(* IEC 61131-3 sources: GradProject/LadderLogic, 14 files *)

(* ---- Test10.st ---- *)
PROGRAM Test_Program
  VAR
    ESP0 AT %QX0.0 : BOOL;
  END_VAR
  VAR
    TMP : BOOL;
  END_VAR
  VAR
    ESP1 AT %QX0.1 : BOOL;
  END_VAR
  VAR
    TMP2 : BOOL;
    TMP4 : BOOL;
    TMP3 : BOOL;
    T0 : TOF;
    TON1 : TON;
    TON2 : TON;
    TON3 : TON;
  END_VAR

  T0(IN := NOT(TMP), PT := T#10000ms);
  ESP0 := T0.Q;
  TON1(IN := ESP0, PT := T#10000ms);
  ESP1 := TON1.Q;
  TON2(IN := ESP1, PT := T#10000ms);
  IF TON2.Q THEN
    ESP1 := FALSE; (*reset*)
  END_IF;
  TMP4 := NOT(TMP3);
  TON3(IN := TMP4, PT := T#30000ms);
  IF TON3.Q THEN
    ESP0 := FALSE; (*reset*)
  END_IF;
END_PROGRAM

CONFIGURATION Config0

  RESOURCE Res0 ON PLC
    TASK MyTask(INTERVAL := T#50ms,PRIORITY := 0);
    PROGRAM instance0 WITH MyTask : Test_Program;
  END_RESOURCE
END_CONFIGURATION

(* ---- Test11\.st ---- *)
PROGRAM Test_Program
  VAR
    ESP0 AT %QX0.0 : BOOL;
    TMP AT %QX1.3 : BOOL;
    ESP1 AT %QX0.1 : BOOL;
  END_VAR
  VAR
    TMP2 : BOOL;
    TMP4 : BOOL;
    TMP3 : BOOL;
    T0 : TOF;
    TON1 : TON;
    TON2 : TON;
    TON3 : TON;
  END_VAR

  T0(IN := TMP, PT := T#10000ms);
  ESP0 := T0.Q;
  TON1(IN := ESP0, PT := T#10000ms);
  ESP1 := TON1.Q;
  TON2(IN := ESP1, PT := T#10000ms);
  IF TON2.Q THEN
    ESP1 := FALSE; (*reset*)
  END_IF;
  TMP4 := NOT(TMP3);
  TON3(IN := TMP4, PT := T#30000ms);
  IF TON3.Q THEN
    ESP0 := FALSE; (*reset*)
  END_IF;
END_PROGRAM

CONFIGURATION Config0

  RESOURCE Res0 ON PLC
    TASK MyTask(INTERVAL := T#50ms,PRIORITY := 0);
    PROGRAM instance0 WITH MyTask : Test_Program;
  END_RESOURCE
END_CONFIGURATION

(* ---- Test12.st ---- *)
PROGRAM Test_Program
  VAR
    ESP0 AT %QX0.0 : BOOL;
    TMP AT %QX0.3 : BOOL;
    ESP1 AT %QX0.1 : BOOL;
  END_VAR
  VAR
    TMP2 : BOOL;
    TMP4 : BOOL;
    TMP3 : BOOL;
    TON1 : TON;
    TON2 : TON;
    TON3 : TON;
  END_VAR

  ESP0 := TMP;
  TON1(IN := ESP0, PT := T#10000ms);
  ESP1 := TON1.Q;
  TON2(IN := ESP1, PT := T#10000ms);
  IF TON2.Q THEN
    ESP1 := FALSE; (*reset*)
  END_IF;
  TMP4 := NOT(TMP3);
  TON3(IN := TMP4, PT := T#30000ms);
  IF TON3.Q THEN
    ESP0 := FALSE; (*reset*)
  END_IF;
END_PROGRAM

CONFIGURATION Config0

  RESOURCE Res0 ON PLC
    TASK MyTask(INTERVAL := T#50ms,PRIORITY := 0);
    PROGRAM instance0 WITH MyTask : Test_Program;
  END_RESOURCE
END_CONFIGURATION

(* ---- Test14.st ---- *)
PROGRAM Test_Program
  VAR
    ESP0 AT %QX0.0 : BOOL;
    TMP AT %QX0.2 : BOOL;
    ESP1 AT %QX0.1 : BOOL;
  END_VAR
  VAR
    TMP2 : BOOL;
    TMP4 : BOOL;
    TMP3 : BOOL;
    TON1 : TON;
    TON2 : TON;
    TON3 : TON;
  END_VAR

  ESP0 := TMP;
  TON1(IN := ESP0, PT := T#10000ms);
  ESP1 := TON1.Q;
  TON2(IN := ESP1, PT := T#10000ms);
  IF TON2.Q THEN
    ESP1 := FALSE; (*reset*)
  END_IF;
  TMP4 := NOT(TMP3);
  TON3(IN := TMP4, PT := T#30000ms);
  IF TON3.Q THEN
    ESP0 := FALSE; (*reset*)
  END_IF;
END_PROGRAM

CONFIGURATION Config0

  RESOURCE Res0 ON PLC
    TASK MyTask(INTERVAL := T#50ms,PRIORITY := 0);
    PROGRAM instance0 WITH MyTask : Test_Program;
  END_RESOURCE
END_CONFIGURATION

(* ---- Test16.st ---- *)
PROGRAM Test_Program
  VAR
    ESP0 AT %QX0.0 : BOOL;
    TMP AT %QX0.2 : BOOL;
    ESP1 AT %QX0.1 : BOOL;
  END_VAR
  VAR
    TMP2 : BOOL;
    TMP4 : BOOL;
    TMP3 : BOOL;
    TON1 : TON;
    TON2 : TON;
  END_VAR

  ESP0 := NOT(TMP);
  TON1(IN := ESP0, PT := T#10000ms);
  ESP1 := TON1.Q;
  TON2(IN := ESP1, PT := T#10000ms);
  IF TON2.Q THEN
    ESP1 := FALSE; (*reset*)
  END_IF;
END_PROGRAM

CONFIGURATION Config0

  RESOURCE Res0 ON PLC
    TASK MyTask(INTERVAL := T#50ms,PRIORITY := 0);
    PROGRAM instance0 WITH MyTask : Test_Program;
  END_RESOURCE
END_CONFIGURATION

(* ---- Test18.st ---- *)
PROGRAM Test_Program
  VAR
    ESP0 AT %QX0.0 : BOOL;
    TMP AT %QX0.2 : BOOL;
    ESP1 AT %QX0.1 : BOOL;
  END_VAR
  VAR
    TMP2 : BOOL;
    TMP4 : BOOL;
    TMP3 : BOOL;
    TON1 : TON;
    TOF0 : TOF;
  END_VAR

  ESP0 := NOT(TMP);
  TON1(IN := ESP0, PT := T#10000ms);
  IF TON1.Q THEN
    ESP0 := FALSE; (*reset*)
  END_IF;
  TOF0(IN := TON1.Q, PT := T#5000ms);
END_PROGRAM

CONFIGURATION Config0

  RESOURCE Res0 ON PLC
    TASK MyTask(INTERVAL := T#50ms,PRIORITY := 0);
    PROGRAM instance0 WITH MyTask : Test_Program;
  END_RESOURCE
END_CONFIGURATION

(* ---- Test19.st ---- *)
PROGRAM Test_Program
  VAR
    ESP0 AT %QX0.0 : BOOL;
    TMP AT %QX0.2 : BOOL;
    ESP1 AT %QX0.1 : BOOL;
  END_VAR
  VAR
    TMP2 : BOOL;
    TMP4 : BOOL;
    TMP3 : BOOL;
    TON1 : TON;
    TOF0 : TOF;
  END_VAR

  TMP := TRUE;
  ESP0 := TMP AND TRUE;
  TON1(IN := ESP0, PT := T#10000ms);
  IF TON1.Q THEN
    ESP0 := FALSE; (*reset*)
  END_IF;
  TOF0(IN := TON1.Q, PT := T#5000ms);
END_PROGRAM

CONFIGURATION Config0

  RESOURCE Res0 ON PLC
    TASK MyTask(INTERVAL := T#50ms,PRIORITY := 0);
    PROGRAM instance0 WITH MyTask : Test_Program;
  END_RESOURCE
END_CONFIGURATION

(* ---- Test20.st ---- *)
PROGRAM Test_Program
  VAR
    ESP0 AT %QX0.0 : BOOL;
    TMP AT %QX0.2 : BOOL;
    ESP1 AT %QX0.1 : BOOL;
  END_VAR
  VAR
    TMP2 : BOOL;
    TMP4 : BOOL;
    TMP3 : BOOL;
    TON1 : TON;
    TOF0 : TOF;
  END_VAR

  TMP := TRUE;
  ESP0 := TRUE;
  TON1(IN := ESP0, PT := T#10000ms);
  IF TON1.Q THEN
    ESP0 := FALSE; (*reset*)
  END_IF;
  TOF0(IN := TON1.Q, PT := T#5000ms);
END_PROGRAM

CONFIGURATION Config0

  RESOURCE Res0 ON PLC
    TASK MyTask(INTERVAL := T#50ms,PRIORITY := 0);
    PROGRAM instance0 WITH MyTask : Test_Program;
  END_RESOURCE
END_CONFIGURATION

(* ---- Test21.st ---- *)
PROGRAM Test_Program
  VAR
    ESP0 AT %QX0.0 : BOOL;
  END_VAR
  VAR
    TMP : BOOL;
  END_VAR
  VAR
    ESP1 AT %QX0.1 : BOOL;
  END_VAR
  VAR
    TON1 : TON;
    TON2 : TON;
  END_VAR

  ESP0 := NOT(TMP);
  TON1(IN := ESP0, PT := T#10000ms);
  ESP1 := TON1.Q;
  TON2(IN := ESP1, PT := T#10000ms);
  IF TON2.Q THEN
    ESP1 := FALSE; (*reset*)
  END_IF;
END_PROGRAM

CONFIGURATION Config0

  RESOURCE Res0 ON PLC
    TASK MyTask(INTERVAL := T#50ms,PRIORITY := 0);
    PROGRAM instance0 WITH MyTask : Test_Program;
  END_RESOURCE
END_CONFIGURATION

(* ---- Test22.st ---- *)
PROGRAM Test_Program
  VAR
    ESP0 AT %QX0.0 : BOOL;
  END_VAR
  VAR
    TMP : BOOL;
  END_VAR
  VAR
    ESP1 AT %QX0.1 : BOOL;
  END_VAR
  VAR
    TON1 : TON;
    TON2 : TON;
  END_VAR

  ESP0 := NOT(TMP);
  TON1(IN := ESP0, PT := T#10000ms);
  ESP1 := TON1.Q;
  TON2(IN := ESP1, PT := T#10000ms);
  IF TON2.Q THEN
    ESP1 := FALSE; (*reset*)
  END_IF;
  IF TON2.Q THEN
    ESP0 := FALSE; (*reset*)
  END_IF;
END_PROGRAM

CONFIGURATION Config0

  RESOURCE Res0 ON PLC
    TASK MyTask(INTERVAL := T#50ms,PRIORITY := 0);
    PROGRAM instance0 WITH MyTask : Test_Program;
  END_RESOURCE
END_CONFIGURATION

(* ---- Test28.st ---- *)
PROGRAM Test_Program
  VAR
    ESP0 AT %QX0.0 : BOOL;
  END_VAR
  VAR
    TMP : BOOL;
  END_VAR
  VAR
    TMP0 AT %QX0.2 : BOOL;
    ESP1 AT %QX0.1 : BOOL;
  END_VAR
  VAR
    TON1 : TON;
    TON2 : TON;
  END_VAR

  ESP0 := NOT(TMP) OR TMP0;
  TON1(IN := ESP0 OR ESP0, PT := T#3000ms);
  ESP1 := TON1.Q;
  TON2(IN := ESP1, PT := T#5000ms);
  TMP := TON2.Q;
END_PROGRAM

CONFIGURATION Config0

  RESOURCE Res0 ON PLC
    TASK MyTask(INTERVAL := T#50ms,PRIORITY := 0);
    PROGRAM instance0 WITH MyTask : Test_Program;
  END_RESOURCE
END_CONFIGURATION

(* ---- Test29.st ---- *)
PROGRAM Test_Program
  VAR
    ESP0 AT %QX0.0 : BOOL;
  END_VAR
  VAR
    TMP : BOOL;
  END_VAR
  VAR
    TMP0 AT %QX0.2 : BOOL;
    ESP1 AT %QX0.1 : BOOL;
  END_VAR
  VAR
    TON1 : TON;
    TON2 : TON;
  END_VAR

  ESP0 := NOT(TMP0) AND TMP;
  TON1(IN := ESP0 OR ESP0, PT := T#3000ms);
  ESP1 := TON1.Q;
  TON2(IN := ESP1, PT := T#5000ms);
  TMP := TON2.Q;
END_PROGRAM

CONFIGURATION Config0

  RESOURCE Res0 ON PLC
    TASK MyTask(INTERVAL := T#50ms,PRIORITY := 0);
    PROGRAM instance0 WITH MyTask : Test_Program;
  END_RESOURCE
END_CONFIGURATION

(* ---- Test30.st ---- *)
PROGRAM Test_Program
  VAR
    ESP0 AT %QX0.0 : BOOL;
  END_VAR
  VAR
    TMP : BOOL;
  END_VAR
  VAR
    TMP0 AT %QX0.2 : BOOL;
    ESP1 AT %QX0.1 : BOOL;
  END_VAR

  ESP0 := NOT(TMP0) AND TMP;
END_PROGRAM

CONFIGURATION Config0

  RESOURCE Res0 ON PLC
    TASK MyTask(INTERVAL := T#50ms,PRIORITY := 0);
    PROGRAM instance0 WITH MyTask : Test_Program;
  END_RESOURCE
END_CONFIGURATION

(* ---- Test31.st ---- *)
PROGRAM Test_Program
  VAR
    ESP0 AT %QX0.0 : BOOL;
  END_VAR
  VAR
    TMP : BOOL;
  END_VAR
  VAR
    TMP0 AT %QX0.2 : BOOL;
    ESP1 AT %QX0.1 : BOOL;
  END_VAR

  ESP0 := NOT(TMP) AND TMP0;
END_PROGRAM

CONFIGURATION Config0

  RESOURCE Res0 ON PLC
    TASK MyTask(INTERVAL := T#50ms,PRIORITY := 0);
    PROGRAM instance0 WITH MyTask : Test_Program;
  END_RESOURCE
END_CONFIGURATION
